// SIMATIC S7-200 SMART project (STEP 7-Micro/WIN SMART), CPU ST60

SYMBOL_TABLE 表格 1
主除尘              V0.0     // 五层96-4
辅助除尘             V0.1     // 一层96-4
仓顶收尘             V0.2     // 在输出点确定启动几个
离心坡              V0.3
反击破              V0.4
v5812            V0.5     // 启动时间12s
双转子              V0.6
二层圆振筛            V0.7     // 启动时间15S
提升机1             V1.0
提升机二             V1.1
小设备              V1.2
圆振筛三层            V1.3
螺旋输送3层           V1.4
圆振筛四层            V1.5
刮板机              V1.6
外部两提升机开启         V1.7
空气斜槽电机1          V2.0
空气斜槽电机2          V2.1
一号皮带启动           V2.2
二号皮带启动           V2.3
END_SYMBOL_TABLE

SYMBOL_TABLE 系统符号
Always_On        SM0.0    // 始终接通
First_Scan_On    SM0.1    // 仅在第一个扫描周期时接通
END_SYMBOL_TABLE

ORGANIZATION_BLOCK MAIN:OB1
TITLE=程序注释
VAR
模式选择:BYTE;	// LB0  0 1 2 3 4 5 分别对应六种模式
圆振筛、提升机选择:BOOL;	// L1.0 
启动:BOOL;	// L1.1 
停止:BOOL;	// L1.2 
皮带选择:BYTE;	// LB2 
停止完成:BOOL;	// L3.0 
提升机开否:BOOL;	// L3.1 
END_VAR
BEGIN
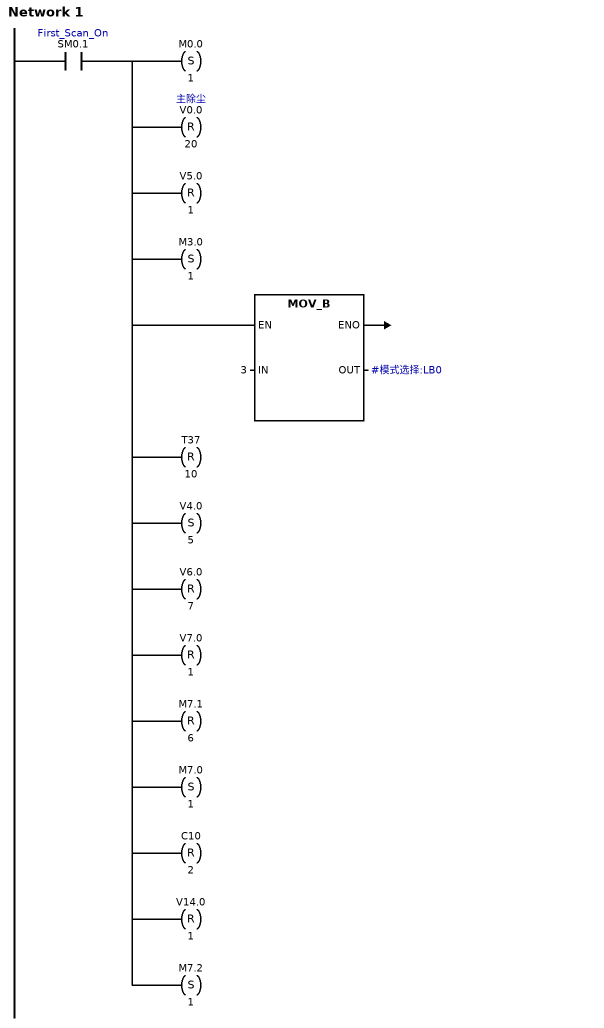
Network 1
LD     First_Scan_On:SM0.1
S      M0.0, 1
R      主除尘:V0.0, 20
R      V5.0, 1
S      M3.0, 1
MOVB   3, #模式选择:LB0
R      T37, 10
S      V4.0, 5
R      V6.0, 7
R      V7.0, 1
R      M7.1, 6
S      M7.0, 1
R      C10, 2
R      V14.0, 1
S      M7.2, 1
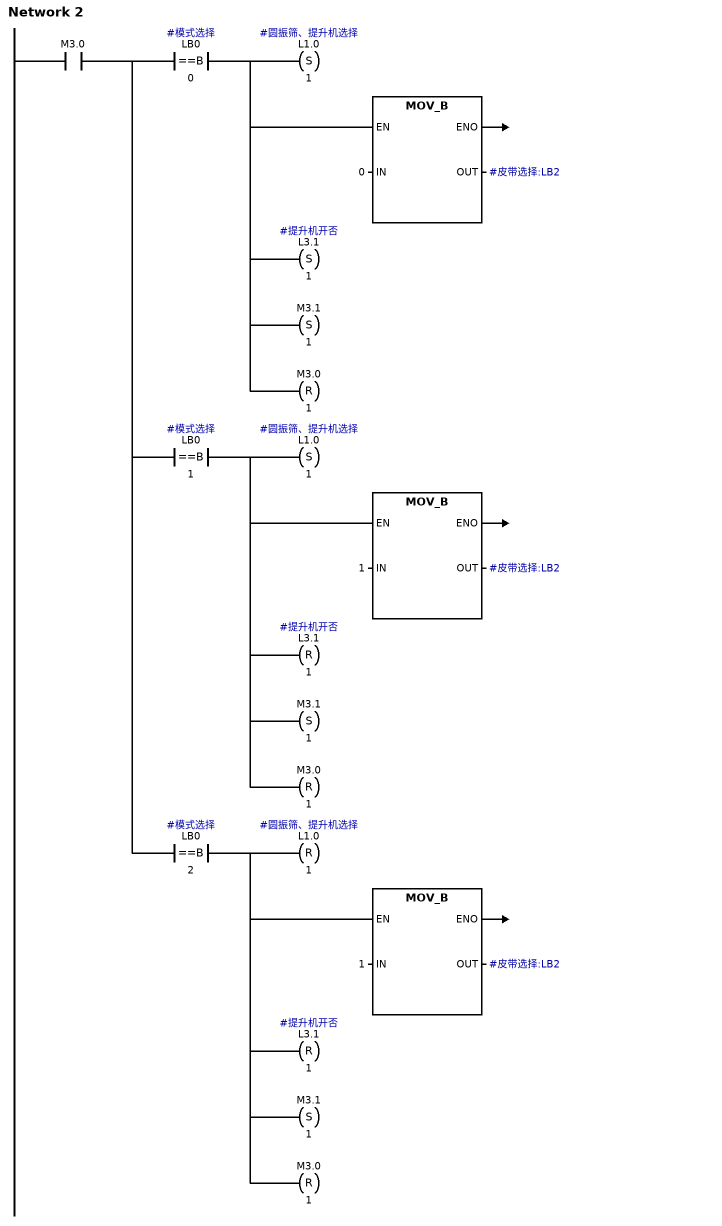
Network 2
LD     M3.0
LPS
AB=    #模式选择:LB0, 0
S      #圆振筛、提升机选择:L1.0, 1
MOVB   0, #皮带选择:LB2
S      #提升机开否:L3.1, 1
S      M3.1, 1
R      M3.0, 1
LRD
AB=    #模式选择:LB0, 1
S      #圆振筛、提升机选择:L1.0, 1
MOVB   1, #皮带选择:LB2
R      #提升机开否:L3.1, 1
S      M3.1, 1
R      M3.0, 1
LPP
AB=    #模式选择:LB0, 2
R      #圆振筛、提升机选择:L1.0, 1
MOVB   1, #皮带选择:LB2
R      #提升机开否:L3.1, 1
S      M3.1, 1
R      M3.0, 1
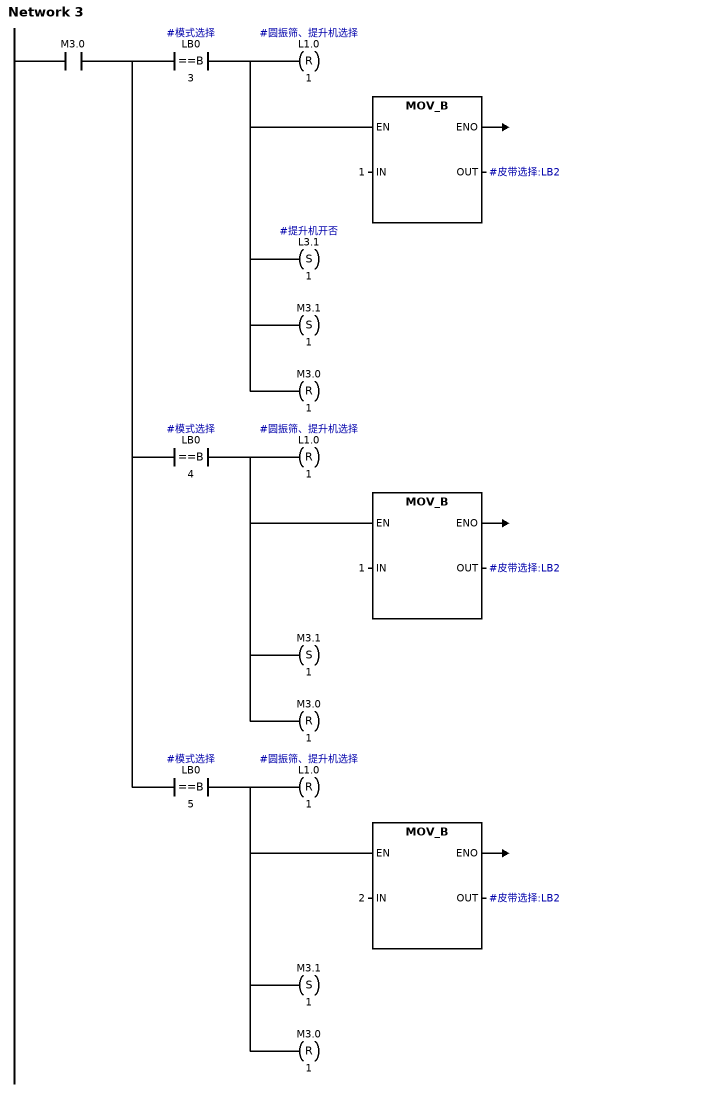
Network 3
LD     M3.0
LPS
AB=    #模式选择:LB0, 3
R      #圆振筛、提升机选择:L1.0, 1
MOVB   1, #皮带选择:LB2
S      #提升机开否:L3.1, 1
S      M3.1, 1
R      M3.0, 1
LRD
AB=    #模式选择:LB0, 4
R      #圆振筛、提升机选择:L1.0, 1
MOVB   1, #皮带选择:LB2
S      M3.1, 1
R      M3.0, 1
LPP
AB=    #模式选择:LB0, 5
R      #圆振筛、提升机选择:L1.0, 1
MOVB   2, #皮带选择:LB2
S      M3.1, 1
R      M3.0, 1
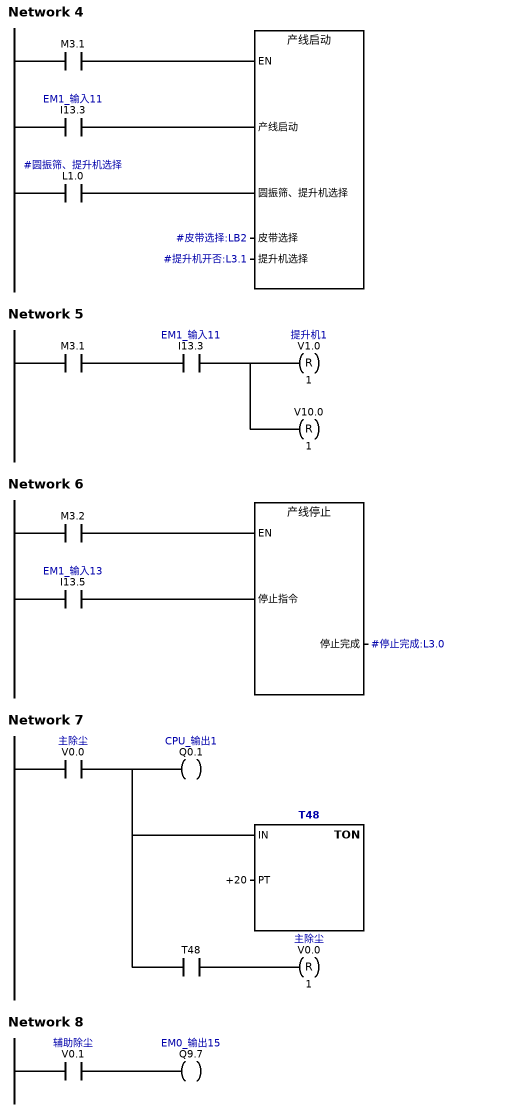
Network 4
LD     M3.1
=      L60.0
LD     EM1_输入11:I13.3
=      L63.7
LD     #圆振筛、提升机选择:L1.0
=      L63.6
LD     L60.0
CALL   产线启动:SBR6, L63.7, L63.6, #皮带选择:LB2, #提升机开否:L3.1
Network 5
LD     M3.1
A      EM1_输入11:I13.3
R      提升机1:V1.0, 1
R      V10.0, 1
Network 6
LD     M3.2
=      L60.0
LD     EM1_输入13:I13.5
=      L63.7
LD     L60.0
CALL   产线停止:SBR7, L63.7, #停止完成:L3.0
Network 7
LD     主除尘:V0.0
=      CPU_输出1:Q0.1
TON    T48, +20
A      T48
R      主除尘:V0.0, 1
Network 8
LD     辅助除尘:V0.1
=      EM0_输出15:Q9.7
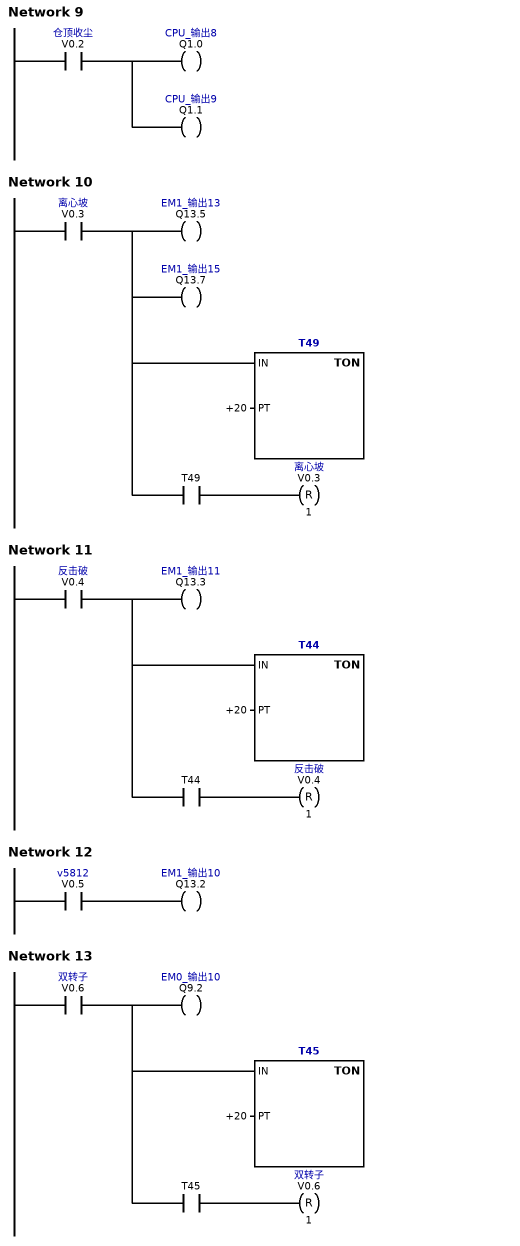
Network 9
LD     仓顶收尘:V0.2
=      CPU_输出8:Q1.0
=      CPU_输出9:Q1.1
Network 10
LD     离心坡:V0.3
=      EM1_输出13:Q13.5
=      EM1_输出15:Q13.7
TON    T49, +20
A      T49
R      离心坡:V0.3, 1
Network 11
LD     反击破:V0.4
=      EM1_输出11:Q13.3
TON    T44, +20
A      T44
R      反击破:V0.4, 1
Network 12
LD     v5812:V0.5
=      EM1_输出10:Q13.2
Network 13
LD     双转子:V0.6
=      EM0_输出10:Q9.2
TON    T45, +20
A      T45
R      双转子:V0.6, 1
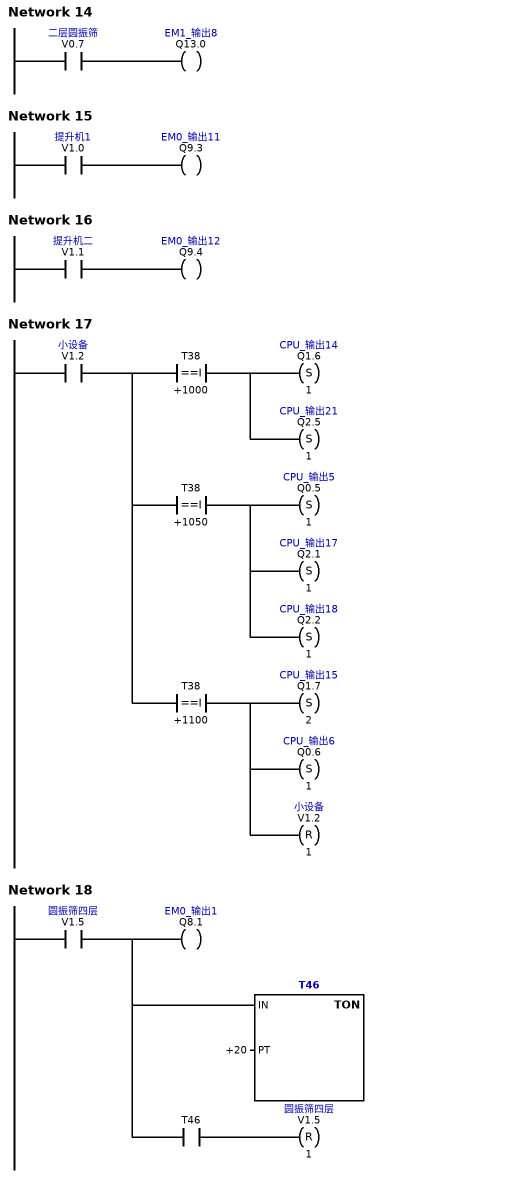
Network 14
LD     二层圆振筛:V0.7
=      EM1_输出8:Q13.0
Network 15
LD     提升机1:V1.0
=      EM0_输出11:Q9.3
Network 16
LD     提升机二:V1.1
=      EM0_输出12:Q9.4
Network 17
LD     小设备:V1.2
LPS
AW=    T38, +1000
S      CPU_输出14:Q1.6, 1
S      CPU_输出21:Q2.5, 1
LRD
AW=    T38, +1050
S      CPU_输出5:Q0.5, 1
S      CPU_输出17:Q2.1, 1
S      CPU_输出18:Q2.2, 1
LPP
AW=    T38, +1100
S      CPU_输出15:Q1.7, 2
S      CPU_输出6:Q0.6, 1
R      小设备:V1.2, 1
Network 18
LD     圆振筛四层:V1.5
=      EM0_输出1:Q8.1
TON    T46, +20
A      T46
R      圆振筛四层:V1.5, 1
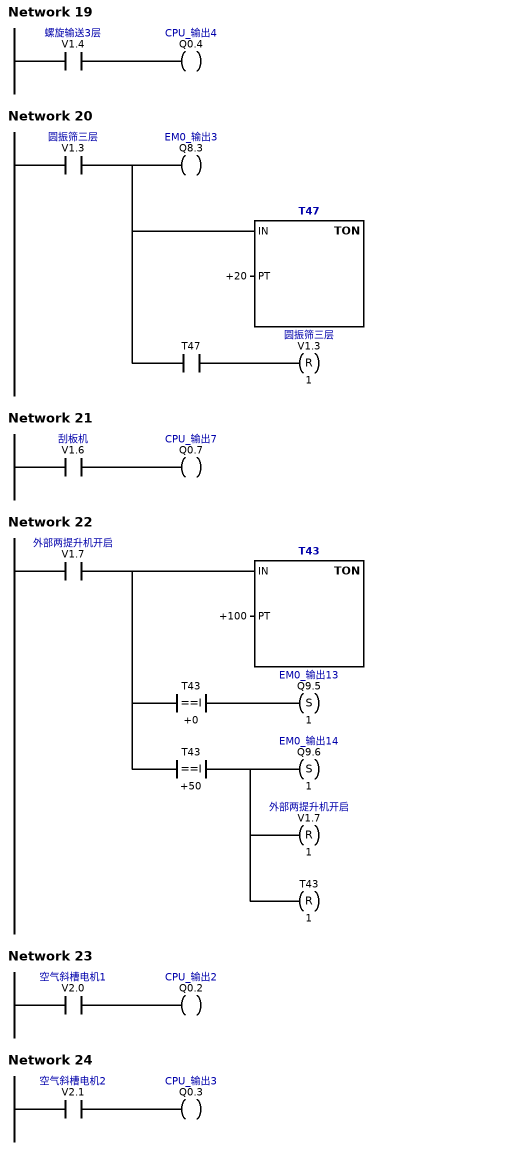
Network 19
LD     螺旋输送3层:V1.4
=      CPU_输出4:Q0.4
Network 20
LD     圆振筛三层:V1.3
=      EM0_输出3:Q8.3
TON    T47, +20
A      T47
R      圆振筛三层:V1.3, 1
Network 21
LD     刮板机:V1.6
=      CPU_输出7:Q0.7
Network 22
LD     外部两提升机开启:V1.7
LPS
TON    T43, +100
AW=    T43, +0
S      EM0_输出13:Q9.5, 1
LPP
AW=    T43, +50
S      EM0_输出14:Q9.6, 1
R      外部两提升机开启:V1.7, 1
R      T43, 1
Network 23
LD     空气斜槽电机1:V2.0
=      CPU_输出2:Q0.2
Network 24
LD     空气斜槽电机2:V2.1
=      CPU_输出3:Q0.3
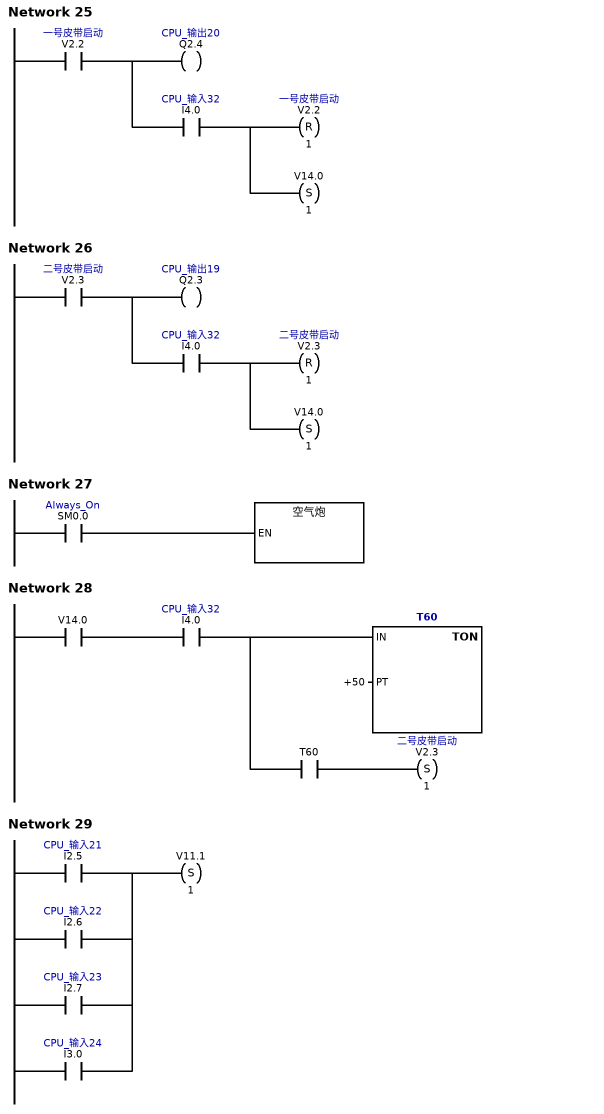
Network 25
LD     一号皮带启动:V2.2
=      CPU_输出20:Q2.4
A      CPU_输入32:I4.0
R      一号皮带启动:V2.2, 1
S      V14.0, 1
Network 26
LD     二号皮带启动:V2.3
=      CPU_输出19:Q2.3
A      CPU_输入32:I4.0
R      二号皮带启动:V2.3, 1
S      V14.0, 1
Network 27
LD     Always_On:SM0.0
CALL   空气炮:SBR0
Network 28
LD     V14.0
A      CPU_输入32:I4.0
TON    T60, +50
A      T60
S      二号皮带启动:V2.3, 1
Network 29
LD     CPU_输入21:I2.5
O      CPU_输入22:I2.6
O      CPU_输入23:I2.7
O      CPU_输入24:I3.0
S      V11.1, 1
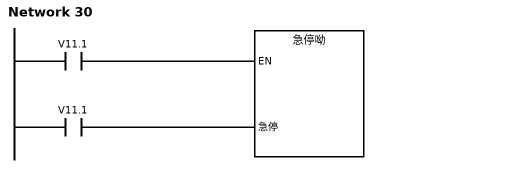
Network 30
LD     V11.1
=      L60.0
LD     V11.1
=      L63.7
LD     L60.0
CALL   急停呦:SBR8, L63.7
END_ORGANIZATION_BLOCK

SUBROUTINE_BLOCK 空气炮:SBR0
TITLE=子程序注释
BEGIN
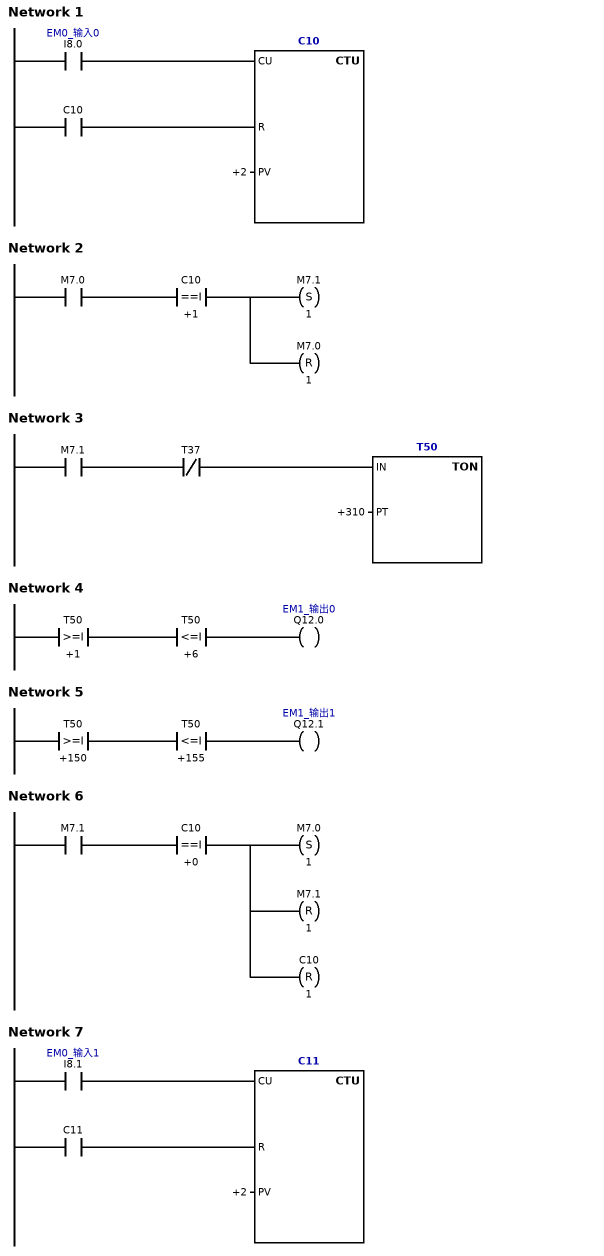
Network 1
LD     EM0_输入0:I8.0
LD     C10
CTU    C10, +2
Network 2
LD     M7.0
AW=    C10, +1
S      M7.1, 1
R      M7.0, 1
Network 3
LD     M7.1
AN     T37
TON    T50, +310
Network 4
LDW>=  T50, +1
AW<=   T50, +6
=      EM1_输出0:Q12.0
Network 5
LDW>=  T50, +150
AW<=   T50, +155
=      EM1_输出1:Q12.1
Network 6
LD     M7.1
AW=    C10, +0
S      M7.0, 1
R      M7.1, 1
R      C10, 1
Network 7
LD     EM0_输入1:I8.1
LD     C11
CTU    C11, +2
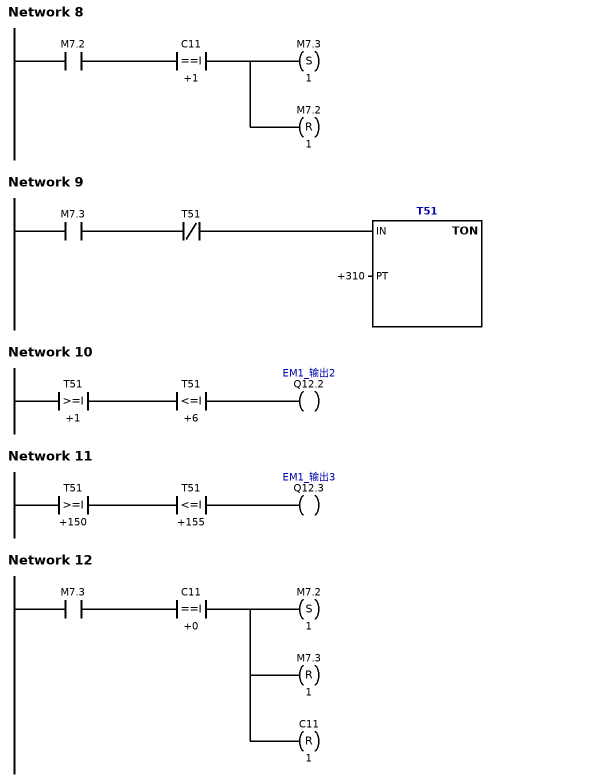
Network 8
LD     M7.2
AW=    C11, +1
S      M7.3, 1
R      M7.2, 1
Network 9
LD     M7.3
AN     T51
TON    T51, +310
Network 10
LDW>=  T51, +1
AW<=   T51, +6
=      EM1_输出2:Q12.2
Network 11
LDW>=  T51, +150
AW<=   T51, +155
=      EM1_输出3:Q12.3
Network 12
LD     M7.3
AW=    C11, +0
S      M7.2, 1
R      M7.3, 1
R      C11, 1
END_SUBROUTINE_BLOCK

SUBROUTINE_BLOCK 除尘启动:SBR1
TITLE=除尘系统
VAR_INPUT
除尘启动:BOOL;	// L0.0 
END_VAR
VAR_OUTPUT
除尘启动完毕:BOOL;	// L0.1 
END_VAR
BEGIN
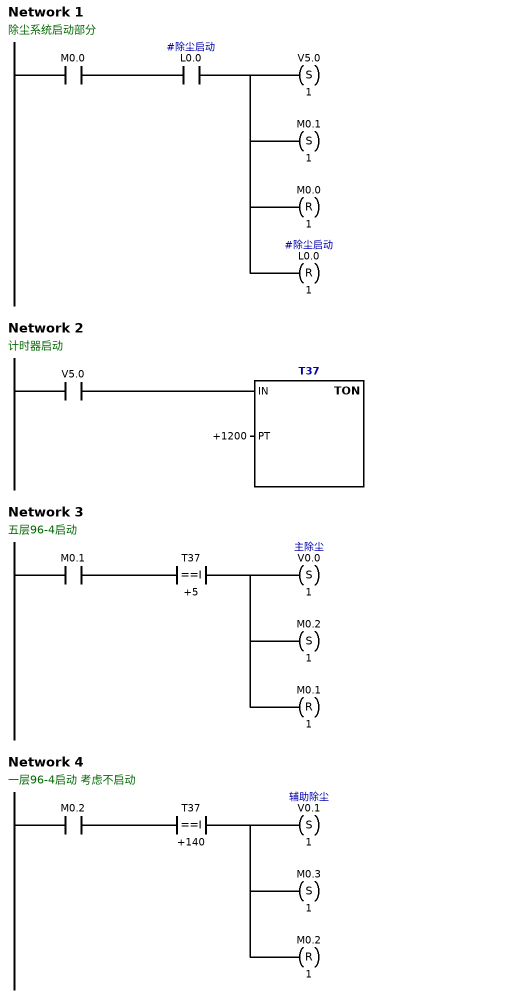
Network 1
// 除尘系统启动部分
LD     M0.0
A      #除尘启动:L0.0
S      V5.0, 1
S      M0.1, 1
R      M0.0, 1
R      #除尘启动:L0.0, 1
Network 2
// 计时器启动
LD     V5.0
TON    T37, +1200
Network 3
// 五层96-4启动
LD     M0.1
AW=    T37, +5
S      主除尘:V0.0, 1
S      M0.2, 1
R      M0.1, 1
Network 4
// 一层96-4启动 考虑不启动
LD     M0.2
AW=    T37, +140
S      辅助除尘:V0.1, 1
S      M0.3, 1
R      M0.2, 1
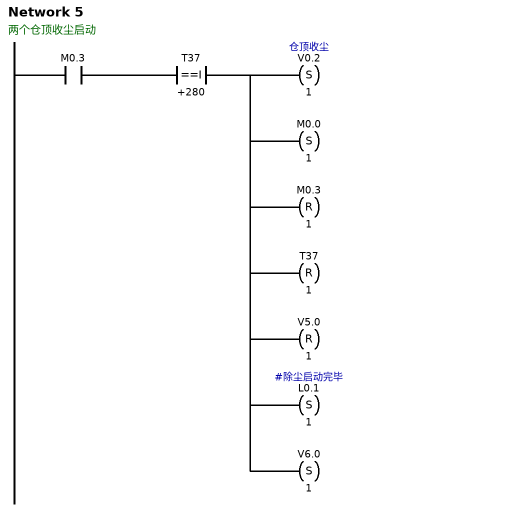
Network 5
// 两个仓顶收尘启动
LD     M0.3
AW=    T37, +280
S      仓顶收尘:V0.2, 1
S      M0.0, 1
R      M0.3, 1
R      T37, 1
R      V5.0, 1
S      #除尘启动完毕:L0.1, 1
S      V6.0, 1
END_SUBROUTINE_BLOCK

SUBROUTINE_BLOCK 必开部分:SBR2
TITLE=什么是必开呢？就是必须要开啊
VAR_INPUT
必开启动:BOOL;	// L0.0 
END_VAR
VAR_OUTPUT
必开启动完毕:BOOL;	// L0.1 
END_VAR
BEGIN
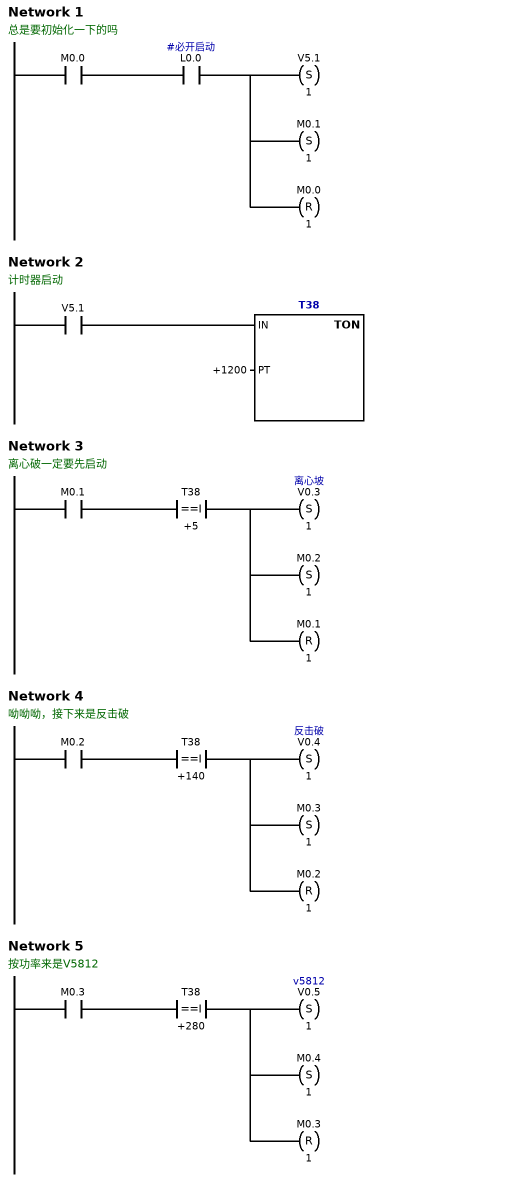
Network 1
// 总是要初始化一下的吗
LD     M0.0
A      #必开启动:L0.0
S      V5.1, 1
S      M0.1, 1
R      M0.0, 1
Network 2
// 计时器启动
LD     V5.1
TON    T38, +1200
Network 3
// 离心破一定要先启动
LD     M0.1
AW=    T38, +5
S      离心坡:V0.3, 1
S      M0.2, 1
R      M0.1, 1
Network 4
// 呦呦呦，接下来是反击破
LD     M0.2
AW=    T38, +140
S      反击破:V0.4, 1
S      M0.3, 1
R      M0.2, 1
Network 5
// 按功率来是V5812
LD     M0.3
AW=    T38, +280
S      v5812:V0.5, 1
S      M0.4, 1
R      M0.3, 1
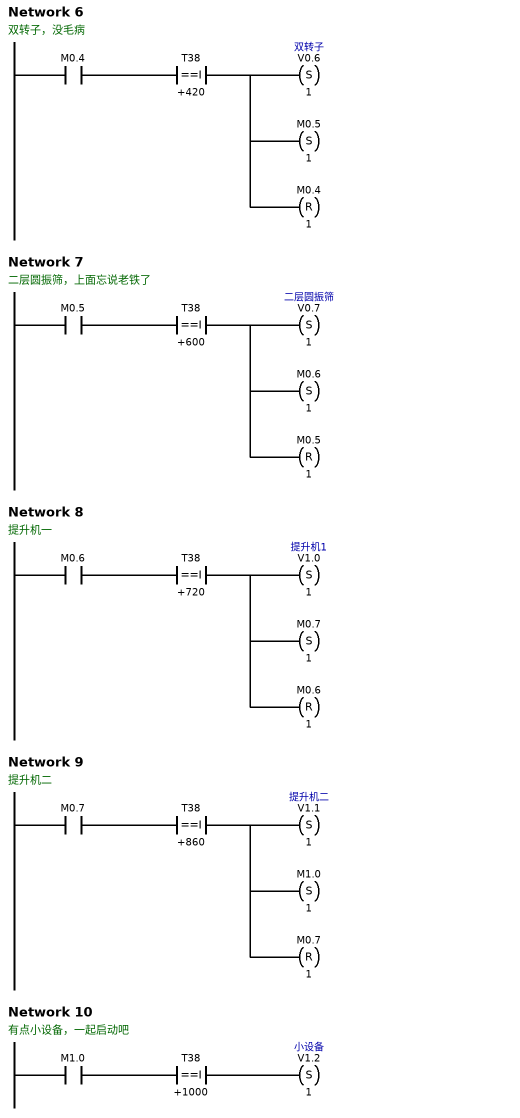
Network 6
// 双转子，没毛病
LD     M0.4
AW=    T38, +420
S      双转子:V0.6, 1
S      M0.5, 1
R      M0.4, 1
Network 7
// 二层圆振筛，上面忘说老铁了
LD     M0.5
AW=    T38, +600
S      二层圆振筛:V0.7, 1
S      M0.6, 1
R      M0.5, 1
Network 8
// 提升机一
LD     M0.6
AW=    T38, +720
S      提升机1:V1.0, 1
S      M0.7, 1
R      M0.6, 1
Network 9
// 提升机二
LD     M0.7
AW=    T38, +860
S      提升机二:V1.1, 1
S      M1.0, 1
R      M0.7, 1
Network 10
// 有点小设备，一起启动吧
LD     M1.0
AW=    T38, +1000
S      小设备:V1.2, 1
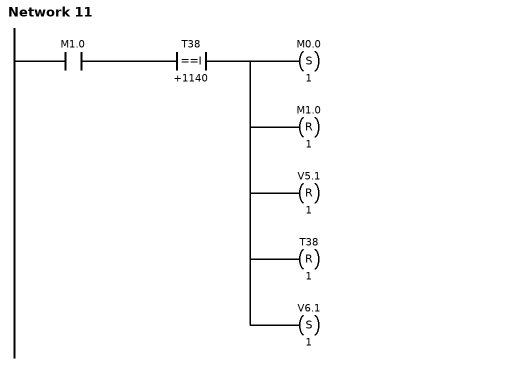
Network 11
LD     M1.0
AW=    T38, +1140
S      M0.0, 1
R      M1.0, 1
R      V5.1, 1
R      T38, 1
S      V6.1, 1
END_SUBROUTINE_BLOCK

SUBROUTINE_BLOCK 圆振筛选择:SBR3
TITLE=子程序注释
VAR_INPUT
圆振筛选择:BOOL;	// L0.0 
圆振筛启动:BOOL;	// L0.1 
END_VAR
VAR_OUTPUT
圆振筛启动完毕:BOOL;	// L0.2 
END_VAR
BEGIN
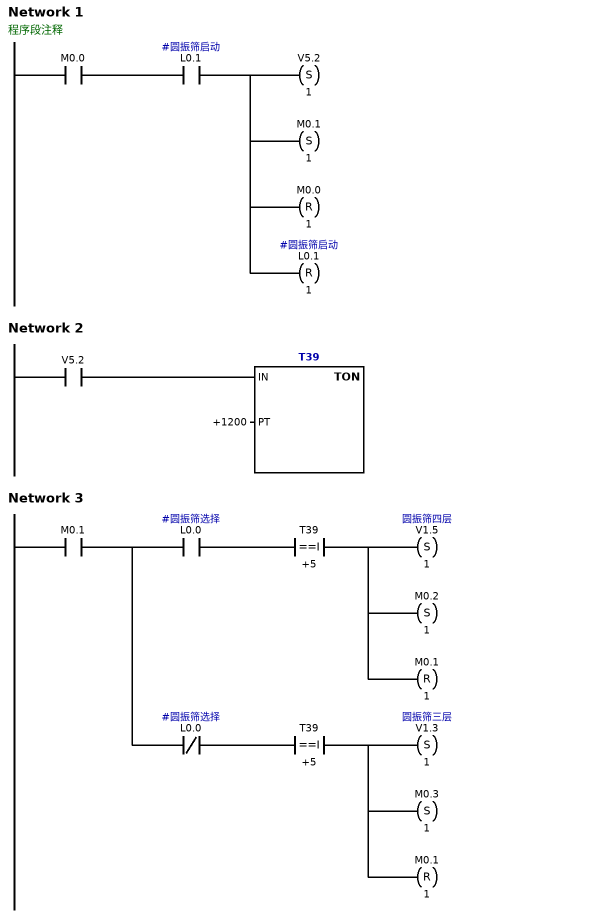
Network 1
// 程序段注释
LD     M0.0
A      #圆振筛启动:L0.1
S      V5.2, 1
S      M0.1, 1
R      M0.0, 1
R      #圆振筛启动:L0.1, 1
Network 2
LD     V5.2
TON    T39, +1200
Network 3
LD     M0.1
LPS
A      #圆振筛选择:L0.0
AW=    T39, +5
S      圆振筛四层:V1.5, 1
S      M0.2, 1
R      M0.1, 1
LPP
AN     #圆振筛选择:L0.0
AW=    T39, +5
S      圆振筛三层:V1.3, 1
S      M0.3, 1
R      M0.1, 1
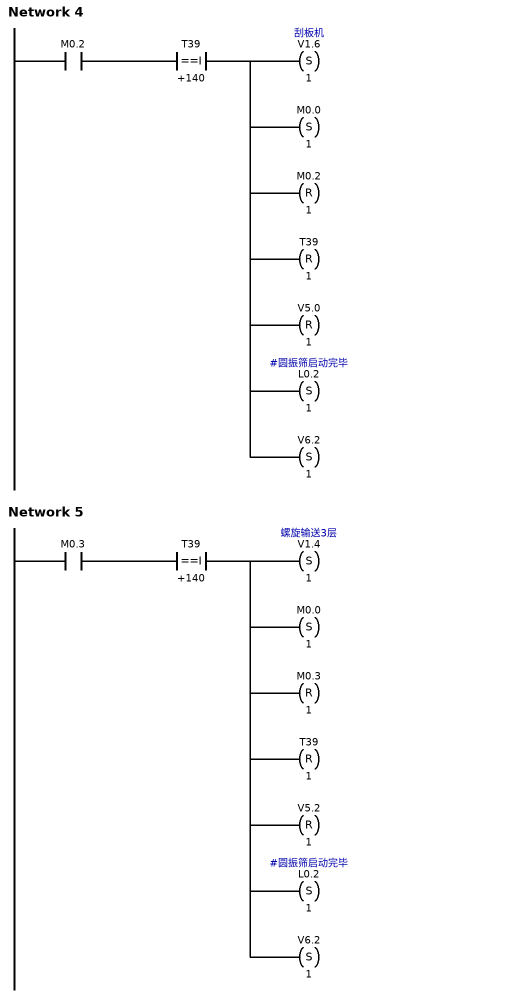
Network 4
LD     M0.2
AW=    T39, +140
S      刮板机:V1.6, 1
S      M0.0, 1
R      M0.2, 1
R      T39, 1
R      V5.0, 1
S      #圆振筛启动完毕:L0.2, 1
S      V6.2, 1
Network 5
LD     M0.3
AW=    T39, +140
S      螺旋输送3层:V1.4, 1
S      M0.0, 1
R      M0.3, 1
R      T39, 1
R      V5.2, 1
S      #圆振筛启动完毕:L0.2, 1
S      V6.2, 1
END_SUBROUTINE_BLOCK

SUBROUTINE_BLOCK 提升机开否:SBR4
TITLE=子程序注释
VAR_INPUT
提升机开否:BOOL;	// L0.0 
提升机启动:BOOL;	// L0.1 
END_VAR
VAR_OUTPUT
提升机部分结束:BOOL;	// L0.2 
END_VAR
BEGIN
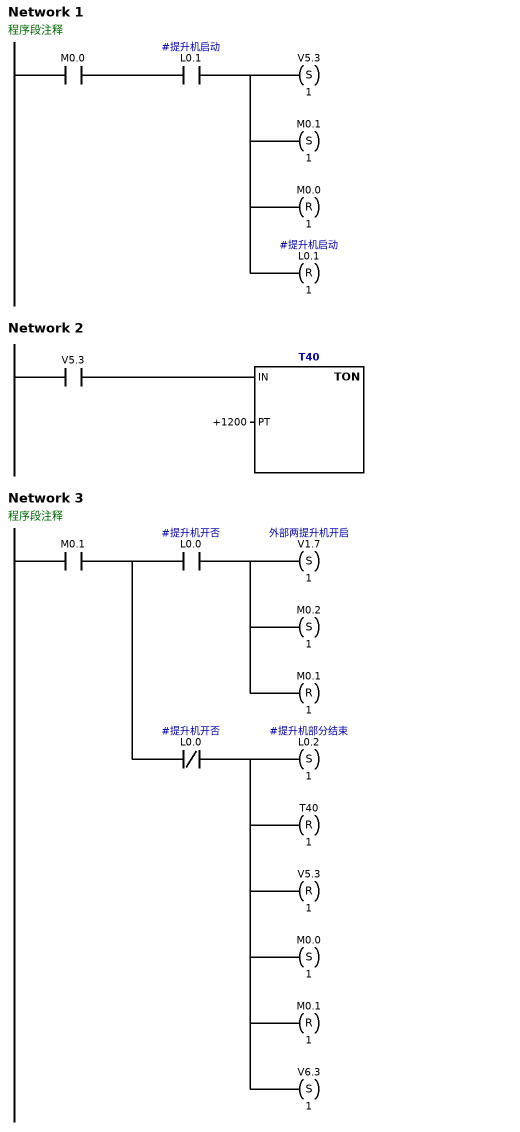
Network 1
// 程序段注释
LD     M0.0
A      #提升机启动:L0.1
S      V5.3, 1
S      M0.1, 1
R      M0.0, 1
R      #提升机启动:L0.1, 1
Network 2
LD     V5.3
TON    T40, +1200
Network 3
// 程序段注释
LD     M0.1
LPS
A      #提升机开否:L0.0
S      外部两提升机开启:V1.7, 1
S      M0.2, 1
R      M0.1, 1
LPP
AN     #提升机开否:L0.0
S      #提升机部分结束:L0.2, 1
R      T40, 1
R      V5.3, 1
S      M0.0, 1
R      M0.1, 1
S      V6.3, 1
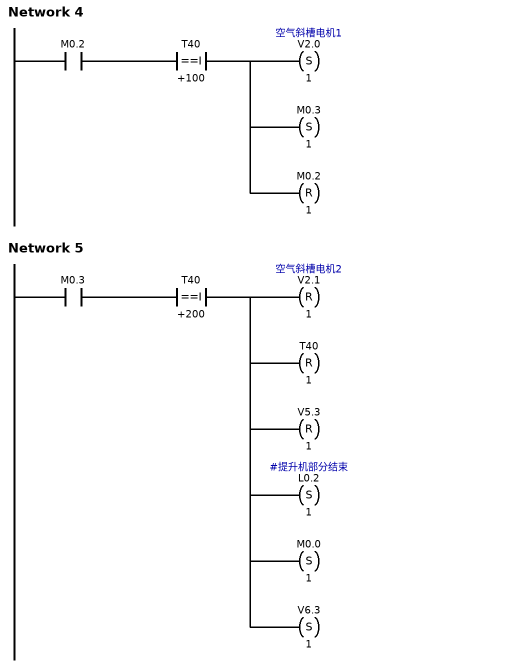
Network 4
LD     M0.2
AW=    T40, +100
S      空气斜槽电机1:V2.0, 1
S      M0.3, 1
R      M0.2, 1
Network 5
LD     M0.3
AW=    T40, +200
R      空气斜槽电机2:V2.1, 1
R      T40, 1
R      V5.3, 1
S      #提升机部分结束:L0.2, 1
S      M0.0, 1
S      V6.3, 1
END_SUBROUTINE_BLOCK

SUBROUTINE_BLOCK 皮带如何:SBR5
TITLE=子程序注释
VAR_INPUT
皮带状态:BYTE;	// LB0 
大皮带启动:BOOL;	// L1.0 
END_VAR
VAR_OUTPUT
大皮带启动完成:BOOL;	// L1.1 
END_VAR
BEGIN
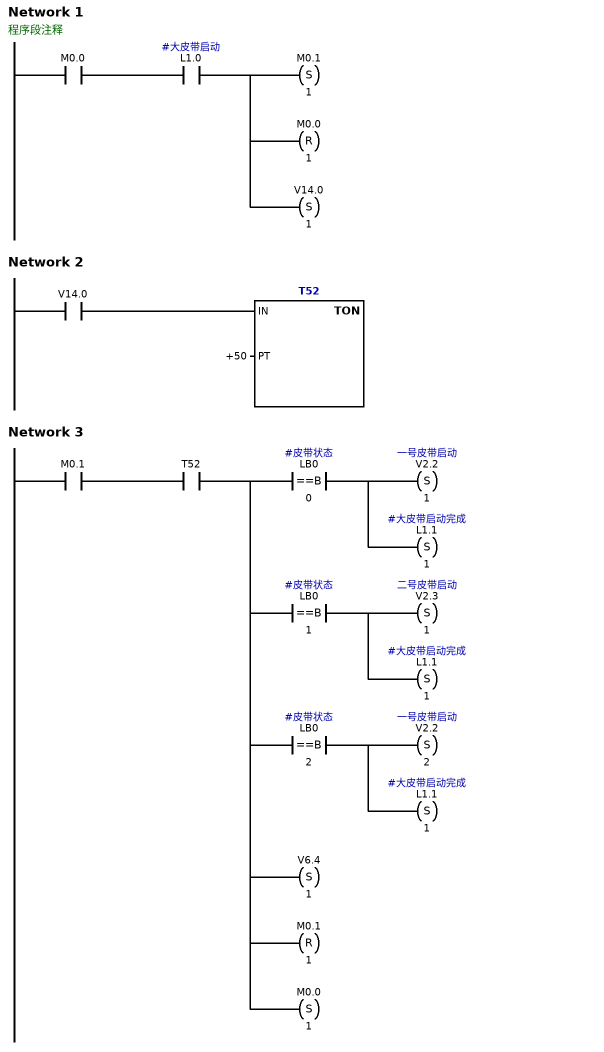
Network 1
// 程序段注释
LD     M0.0
A      #大皮带启动:L1.0
S      M0.1, 1
R      M0.0, 1
S      V14.0, 1
Network 2
LD     V14.0
TON    T52, +50
Network 3
LD     M0.1
A      T52
LPS
AB=    #皮带状态:LB0, 0
S      一号皮带启动:V2.2, 1
S      #大皮带启动完成:L1.1, 1
LRD
AB=    #皮带状态:LB0, 1
S      二号皮带启动:V2.3, 1
S      #大皮带启动完成:L1.1, 1
LRD
AB=    #皮带状态:LB0, 2
S      一号皮带启动:V2.2, 2
S      #大皮带启动完成:L1.1, 1
LPP
S      V6.4, 1
R      M0.1, 1
S      M0.0, 1
END_SUBROUTINE_BLOCK

SUBROUTINE_BLOCK 产线启动:SBR6
TITLE=子程序注释
VAR_INPUT
产线启动:BOOL;	// L0.0 
圆振筛、提升机选择:BOOL;	// L0.1 
皮带选择:BYTE;	// LB1 
提升机选择:BOOL;	// L2.0 
END_VAR
VAR
除尘启动完毕:BOOL;	// L2.1 
必开启动完毕:BOOL;	// L2.2 
圆振筛启动完毕:BOOL;	// L2.3 
提升机启动完毕:BOOL;	// L2.4 
启动完毕:BOOL;	// L2.5 
END_VAR
BEGIN
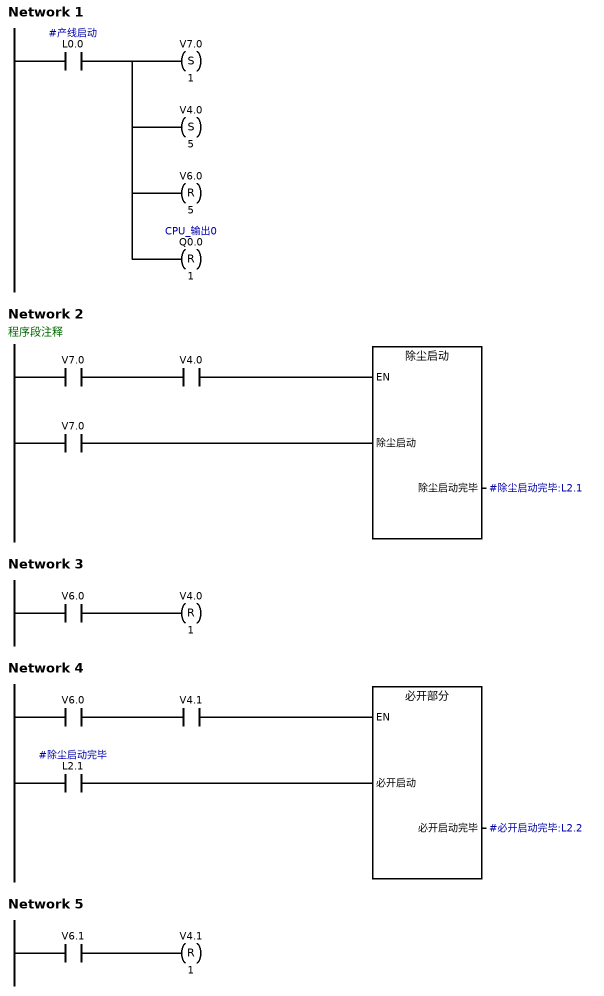
Network 1
LD     #产线启动:L0.0
S      V7.0, 1
S      V4.0, 5
R      V6.0, 5
R      CPU_输出0:Q0.0, 1
Network 2
// 程序段注释
LD     V7.0
A      V4.0
=      L60.0
LD     V7.0
=      L63.7
LD     L60.0
CALL   除尘启动:SBR1, L63.7, #除尘启动完毕:L2.1
Network 3
LD     V6.0
R      V4.0, 1
Network 4
LD     V6.0
A      V4.1
=      L60.0
LD     #除尘启动完毕:L2.1
=      L63.7
LD     L60.0
CALL   必开部分:SBR2, L63.7, #必开启动完毕:L2.2
Network 5
LD     V6.1
R      V4.1, 1
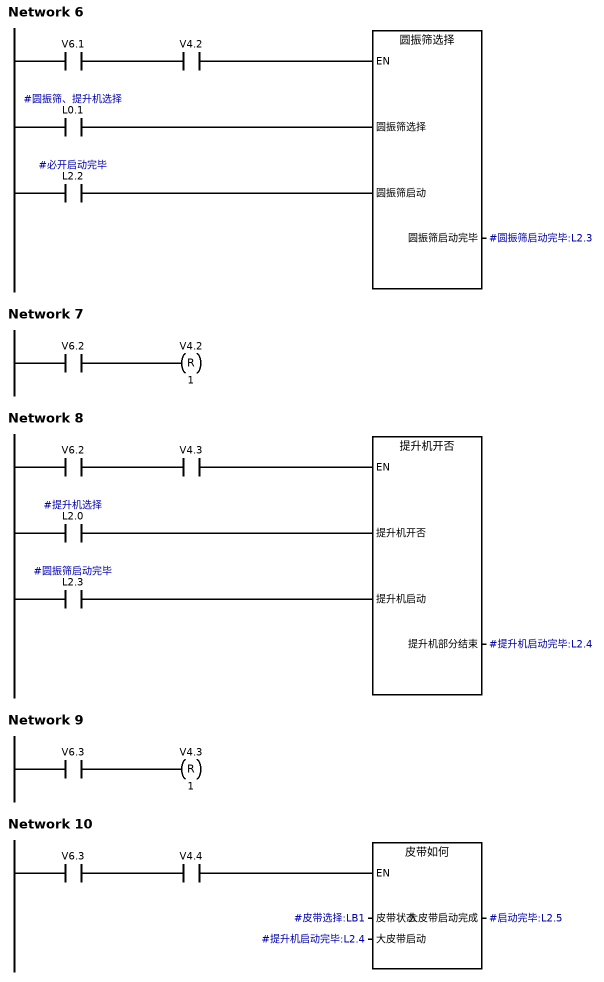
Network 6
LD     V6.1
A      V4.2
=      L60.0
LD     #圆振筛、提升机选择:L0.1
=      L63.7
LD     #必开启动完毕:L2.2
=      L63.6
LD     L60.0
CALL   圆振筛选择:SBR3, L63.7, L63.6, #圆振筛启动完毕:L2.3
Network 7
LD     V6.2
R      V4.2, 1
Network 8
LD     V6.2
A      V4.3
=      L60.0
LD     #提升机选择:L2.0
=      L63.7
LD     #圆振筛启动完毕:L2.3
=      L63.6
LD     L60.0
CALL   提升机开否:SBR4, L63.7, L63.6, #提升机启动完毕:L2.4
Network 9
LD     V6.3
R      V4.3, 1
Network 10
LD     V6.3
A      V4.4
CALL   皮带如何:SBR5, #皮带选择:LB1, #提升机启动完毕:L2.4, #启动完毕:L2.5
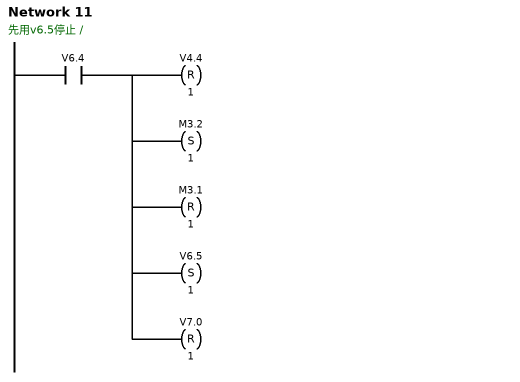
Network 11
// 先用v6.5停止
// 
LD     V6.4
R      V4.4, 1
S      M3.2, 1
R      M3.1, 1
S      V6.5, 1
R      V7.0, 1
END_SUBROUTINE_BLOCK

SUBROUTINE_BLOCK 产线停止:SBR7
TITLE=子程序注释
VAR_INPUT
停止指令:BOOL;	// L0.0 
END_VAR
VAR_OUTPUT
停止完成:BOOL;	// L0.1 
END_VAR
BEGIN
